// TIA Portal V19 export
DATA_BLOCK "A0303_Spalla_Coda"   // DB161
// stored: InstanceOfName A0303_Spalla_FB, InstanceOfType FB
"A0303_Spalla_FB"
   // VAR_INPUT
   //    AreaInterface : "AreaInterface";
   //    ZSI : "udt_ZoneSafetyInterface";
   //    DSI : "udt_DeviceSafetyInterface";
   //    DataIn : Struct
   //       OP_Pos : Bool;
   //       FC_Aticoll_Paregg { ExternalWritable := 'False'} : Bool;
   //    END_STRUCT;
   //    CIn : Struct
   //       Manager : "Positioning_DOL_Machine_Manager";
   //       Antiribaltamento : Struct
   //          OutOfWorkspace : Bool;
   //       END_STRUCT;
   //       Pareggiatore : Struct
   //          ActualPosition : LReal;
   //       END_STRUCT;
   //    END_STRUCT;
   //    Config : Struct
   //       Ax : "Positioning_DOL_Machine_Config";
   //       DelayMissingCondition { ExternalAccessible := 'False'; ExternalVisible := 'False'; ExternalWritable := 'False'} : Time;
   //    END_STRUCT;
   //    HWID : Struct
   //       Ax_TEL1 : HW_SUBMODULE;
   //       Enc_IO : HW_SUBMODULE;
   //    END_STRUCT;
   // END_VAR
   // VAR_OUTPUT
   //    MachineInterface { ExternalAccessible := 'False'; ExternalVisible := 'False'; ExternalWritable := 'False'} : "MachineInterface";
   //    COut : Struct
   //       Ax : "Positioning_DOL_Machine_COut";
   //    END_STRUCT;
   // END_VAR
   // VAR_IN_OUT
   //    Par : Struct
   //       Ax : "Positioning_DOL_Machine_Par";
   //       Ax_Pers : "Positioning_DOL_Machine_Pers_Data";
   //       Enc : "PosFbk_RTN";
   //    END_STRUCT;
   //    Par_Mach : Struct
   //       MinDistanzaConParegg : LReal;
   //       ToleranceWindow : LReal;
   //    END_STRUCT;
   // END_VAR
   // VAR
   //    Alarm : Struct
   //       Ax : "Positioning_DOL_Machine_Alr";
   //       Enc : "PosFbk_Encoder_Alr";
   //    END_STRUCT;
   //    Warning : Struct
   //       Ax : "Positioning_DOL_Machine_Wng";
   //       SW_Limit_AntiCollision : Bool;
   //       OP_POS_MissingCnd : Bool;
   //    END_STRUCT;
   //    HMI : Struct
   //       PbPreset : Bool;
   //       B_Preset_UM2 : Bool;
   //       PresetValue : LReal;
   //    END_STRUCT;
   //    Sts : Struct
   //       AlarmsPresence : Bool;
   //       WarningsPresence : Bool;
   //       OP_CanMoveFreely : Bool;
   //       OP_Pos_Cnd : Bool;
   //    END_STRUCT;
   //    Ctrl : Struct
   //       OP_Pos_Aut : Bool;
   //       OP_Pos_Run : Bool;
   //       OP_Pos_Man : Bool;
   //       OP_Pos : Bool;
   //    END_STRUCT;
   //    Ax : "Positioning_DOL_Machine_FB";
   //    Enc : "PosFbk_SickAFM60";
   //    Enc_ITF : "PosFbk_ITF";
   //    AUX { ExternalAccessible := 'False'; ExternalVisible := 'False'; ExternalWritable := 'False'} : Struct
   //       OP_Pos_PB : Bool;
   //    END_STRUCT;
   //    TON_OP_POS_MissingCnd : IEC_TIMER;
   //    TON_DistanzaOK : IEC_TIMER;
   // END_VAR
BEGIN
END_DATA_BLOCK
